FUNCTION_BLOCK Engine (* Simple FB with one algorithm *)
  (* Standard: 61499-1 *)
  (* Version 1.0, 2025-07-18, vadim *)
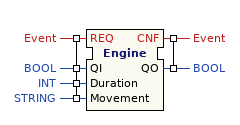
  EVENT_INPUT
    REQ WITH Duration, Movement, QI; (* Normal Execution Request *)
  END_EVENT
  EVENT_OUTPUT
    CNF WITH QO; (* Execution Confirmation *)
  END_EVENT
  VAR_INPUT
    QI : BOOL;
    Duration : INT; (* Duration (ms) *)
    Movement : STRING; (* Kind of movement *)
  END_VAR
  VAR_OUTPUT
    QO : BOOL;
  END_VAR
  EC_STATES
    REQ : REQ -> CNF;
  END_STATES
  ALGORITHM REQ IN ST:

  END_ALGORITHM
END_FUNCTION_BLOCK
